FUNCTION_BLOCK TcaCarrier EXTENDS TcoCore.TcoComponent IMPLEMENTS ITcaCarrier
VAR CONSTANT
	MAX_WORKPIECEPLACES : INT := 127;
END_VAR

VAR PERSISTENT
	_carrierID : INT;	
	_data : TcaCarrierData;
	_config : TcaCarrierConfig;
	_arrayOfWorkpiecePlaces : ARRAY[0..MAX_WORKPIECEPLACES] OF TcaWorkpiecePlace(THIS^);
END_VAR

VAR
	_ModifyTask : TcaCarrierModifyTask(THIS^);	
	_modifyId : INT := 0;
	_i : INT;
		
	_WorkpieceStatusCount : ARRAY[0..eTcaWorkpiecePlaceStatus.MAXSIZE] OF INT;
	_PrimaryStatus : eTcaWorkpiecePlaceStatus;
	_SecondaryStatus : eTcaWorkpiecePlaceStatus;
	_PrimaryStatusCount : INT;
	_SecondaryStatusCount : INT;
	
	_ConfigError	: BOOL;
	
END_VAR

THIS^._ModifyTask(inoArrayOfWorkpiecePlaces := _arrayOfWorkpiecePlaces);

FOR _i:= 0 TO MAX_WORKPIECEPLACES DO
	_arrayOfWorkpiecePlaces[_i]();
END_FOR

METHOD ApplyConfig : REFERENCE TO TcaCarrier
VAR
	tmpData				: TcaCarrierConfig;
	
	tmpOffset 			: REAL;
	tmpOddRow			: INT;
	tmpEvenRow			: INT;
	tmpWorkpieceCount	: INT;
	
	tmpPos		 		: INT;
	tmpLoc		 		: INT;		
	tmpRow 				: INT;
	//tmpLvl				: INT;
	
	nRowNumber			: INT;
	nLocationNumber		: INT; 
	
	ni					: INT;
	
	tmpCoordinate 		: ST_Coordinate;		
END_VAR
tmpData := _config;

CASE tmpData.Layout OF
	eTcaCarrierLayout.Layout1 : 
		tmpOffset := 0;
		tmpOddRow := tmpData.PositionsInRow;
        tmpEvenRow := tmpData.PositionsInRow;
        tmpWorkpieceCount := tmpData.PositionsInRow*tmpData.PositionsInColumn;
		
    eTcaCarrierLayout.Layout2 :
		tmpOffset := 0.5;
		tmpOddRow := tmpData.PositionsInRow;
		tmpEvenRow := tmpData.PositionsInRow;
        tmpWorkpieceCount := tmpData.PositionsInRow*tmpData.PositionsInColumn;
		 
    eTcaCarrierLayout.Layout3 :
		 tmpOffset := -0.5;
		 tmpOddRow := tmpData.PositionsInRow;
         tmpEvenRow := tmpData.PositionsInRow;
         tmpWorkpieceCount := tmpData.PositionsInRow*tmpData.PositionsInColumn;	
		 
	eTcaCarrierLayout.Layout4 :
		 tmpOffset := -0.5;
		 tmpOddRow := tmpData.PositionsInRow;
         tmpEvenRow := tmpData.PositionsInRow + 1;
         tmpWorkpieceCount := tmpData.PositionsInRow*tmpData.PositionsInColumn + tmpData.PositionsInColumn/2;
		
	eTcaCarrierLayout.Layout5 :
		 tmpOffset := 0.5;
		 tmpOddRow := tmpData.PositionsInRow;
         tmpEvenRow := tmpData.PositionsInRow - 1;
         tmpWorkpieceCount := tmpData.PositionsInRow*tmpData.PositionsInColumn - tmpData.PositionsInColumn/2;
		 
END_CASE


MEMSET(ADR(_data.WorkpiecesCoordinate),0,SIZEOF(_data.WorkpiecesCoordinate));
MEMSET(ADR(_data.WorkpiecesEnabled),0,SIZEOF(_data.WorkpiecesEnabled));


FOR ni:= 0 TO tmpWorkpieceCount-1 DO
	
	// Bestimmen des Reihen und Spaltenndex und der x und y-Koordinate
	tmpPos := ni MOD tmpWorkpieceCount;
	tmpRow := tmpPos/(tmpOddRow + tmpEvenRow);	
	tmpLoc := tmpPos MOD (tmpOddRow + tmpEvenRow);
	
	IF tmpLoc >= tmpOddRow THEN
	    // gerade Reihe
	    nRowNumber := tmpRow*2 + 1;
	    nLocationNumber := tmpLoc - tmpOddRow;
	    tmpCoordinate.fX := tmpData.ColumnDistance*(nLocationNumber + tmpOffset)+tmpData.CoordinateFirstWorkpiece.fX;
	    tmpCoordinate.fY := tmpData.RowDistance*nRowNumber+tmpData.CoordinateFirstWorkpiece.fY;
	ELSE
	    // ungerade Reihe
	    nRowNumber := tmpRow*2;
	    nLocationNumber := tmpLoc;
	    tmpCoordinate.fX := tmpData.ColumnDistance*nLocationNumber+tmpData.CoordinateFirstWorkpiece.fX;
	    tmpCoordinate.fY := tmpData.RowDistance*nRowNumber+tmpData.CoordinateFirstWorkpiece.fY;
	END_IF
	
	tmpCoordinate.nOriginId := 0;
		
	_data.WorkpiecesCoordinate[ni] := tmpCoordinate;
	_data.WorkpiecesEnabled[ni] := TRUE;

END_FOR
END_METHOD

METHOD ChangeData : ITcoTaskStatus 
VAR_INPUT
	inData : TcaCarrierData;
END_VAR
ChangeData := _ModifyTask.InvokeCarrierData(inData);
END_METHOD

METHOD ColumnDistance : REFERENCE TO TcaCarrier
VAR_INPUT
	inDistance : LREAL;
END_VAR
THIS^._config.ColumnDistance:= inDistance;
ColumnDistance REF= THIS^;
END_METHOD

METHOD CoordinateFirstWorkpiece : REFERENCE TO TcaCarrier
VAR_INPUT
	inCoordinate : ST_Coordinate;
END_VAR
THIS^._config.CoordinateFirstWorkpiece:= inCoordinate;
CoordinateFirstWorkpiece REF= THIS^;
END_METHOD

METHOD CoordinatesOf : ST_Coordinate
VAR_INPUT
	WorkpiecePlace		: INT;
END_VAR

VAR
	tmpData				: TcaCarrierConfig;
	
	tmpOffset 			: REAL;
	tmpOddRow			: INT;
	tmpEvenRow			: INT;
	tmpWorkpieceCount	: INT;
	
	tmpPos		 		: INT;
	tmpLoc		 		: INT;		
	tmpRow 				: INT;
	//tmpLvl				: INT;
	
	nRowNumber			: INT;
	nLocationNumber		: INT; 
	
	tmpCoordinate 		: ST_Coordinate;		
	
END_VAR
IF WorkpiecePlace = 0 THEN
	RETURN;
END_IF

tmpData := _config;

CASE tmpData.Layout OF
	eTcaCarrierLayout.Layout1 : 
		tmpOffset := 0;
		tmpOddRow := tmpData.PositionsInRow;
        tmpEvenRow := tmpData.PositionsInRow;
        tmpWorkpieceCount := tmpData.PositionsInRow*tmpData.PositionsInColumn;
		
    eTcaCarrierLayout.Layout2 :
		tmpOffset := 0.5;
		tmpOddRow := tmpData.PositionsInRow;
		tmpEvenRow := tmpData.PositionsInRow;
        tmpWorkpieceCount := tmpData.PositionsInRow*tmpData.PositionsInColumn;
		 
    eTcaCarrierLayout.Layout3 :
		 tmpOffset := -0.5;
		 tmpOddRow := tmpData.PositionsInRow;
         tmpEvenRow := tmpData.PositionsInRow;
         tmpWorkpieceCount := tmpData.PositionsInRow*tmpData.PositionsInColumn;	
		 
	eTcaCarrierLayout.Layout4 :
		 tmpOffset := -0.5;
		 tmpOddRow := tmpData.PositionsInRow;
         tmpEvenRow := tmpData.PositionsInRow + 1;
         tmpWorkpieceCount := tmpData.PositionsInRow*tmpData.PositionsInColumn + tmpData.PositionsInColumn/2;
		
	eTcaCarrierLayout.Layout5 :
		 tmpOffset := 0.5;
		 tmpOddRow := tmpData.PositionsInRow;
         tmpEvenRow := tmpData.PositionsInRow - 1;
         tmpWorkpieceCount := tmpData.PositionsInRow*tmpData.PositionsInColumn - tmpData.PositionsInColumn/2;
		 
END_CASE

// Bestimmen des Reihen und Spaltenndex und der x und y-Koordinate
tmpPos := (WorkpiecePlace - 1) MOD tmpWorkpieceCount;
tmpRow := tmpPos/(tmpOddRow + tmpEvenRow);	
tmpLoc := tmpPos MOD (tmpOddRow + tmpEvenRow);
//tmpLvl := (Position - 1)/tmpWorkpieceCount;


IF tmpLoc >= tmpOddRow THEN
    // gerade Reihe
    nRowNumber := tmpRow*2 + 1;
    nLocationNumber := tmpLoc - tmpOddRow;
    tmpCoordinate.fX := tmpData.ColumnDistance*(nLocationNumber + tmpOffset);
    tmpCoordinate.fY := tmpData.RowDistance*nRowNumber;
ELSE
    // ungerade Reihe
    nRowNumber := tmpRow*2;
    nLocationNumber := tmpLoc;
    tmpCoordinate.fX := tmpData.ColumnDistance*nLocationNumber;
    tmpCoordinate.fY := tmpData.RowDistance*nRowNumber;
END_IF
		

//tmpCoordinate.fZ := tmpLvl*fLevelDistance;

// Koordinaten zurückgeben
tmpCoordinate.nOriginId := 0;
CoordinatesOf := tmpCoordinate;
END_METHOD

METHOD CountEmptyPlaces : INT

VAR
	tmp				: INT;
	ni				: INT;
END_VAR
CountEmptyPlaces := 0;

FOR ni := 0 TO MAX_WORKPIECEPLACES DO
	
	IF NOT _arrayOfWorkpiecePlaces[ni].Enabled THEN
		CONTINUE;
	END_IF
	
	IF _arrayOfWorkpiecePlaces[ni].Error THEN
		CONTINUE;
	END_IF

	IF NOT _arrayOfWorkpiecePlaces[ni].WorkpiecePresent THEN
		tmp := tmp + 1;	
	END_IF

END_FOR

CountEmptyPlaces := tmp;
END_METHOD

METHOD CountPlacesByStatus : INT
VAR_INPUT
	nStatus			: INT;
END_VAR

VAR
	tmp				: INT;
	ni				: INT;
END_VAR
CountPlacesByStatus := 0;

FOR ni := 0 TO MAX_WORKPIECEPLACES DO

	IF NOT _data.WorkpiecesData[ni].Enabled THEN
		CONTINUE;
	END_IF	
	
	IF _data.WorkpiecesData[ni].Error THEN
		CONTINUE;
	END_IF

	IF _data.WorkpiecesData[ni].CurrentStatus = nStatus THEN
			tmp := tmp + 1;
	END_IF
	
END_FOR

CountPlacesByStatus := tmp;
END_METHOD

PROPERTY Data : REFERENCE TO TcaCarrierData
GET
Data REF= _data;
END_GET
END_PROPERTY

//FB_Init ist immer implizit verfügbar und wird primär für die Initialisierung verwendet.
//Der Rückgabewert wird nicht ausgewertet. Für gezielte Einflussnahme können Sie
//die Methoden explizit deklarieren und darin mit dem Standard-Initialisierungscode 
//zusätzlichen Code bereitstellen. Sie können den Rückgabewert auswerten.
METHOD FB_Init: BOOL
VAR_INPUT    
bInitRetains: BOOL; // TRUE: Die Retain-Variablen werden initialisiert (Reset warm / Reset kalt)    
bInCopyCode: BOOL;  // TRUE: Die Instanz wird danach in den Kopiercode kopiert (Online-Change)
ParentObject : ITcoObject;
END_VAR
VAR
	_i : INT;
END_VAR
FOR _i:= 0 TO MAX_WORKPIECEPLACES DO
	_arrayOfWorkpiecePlaces[_i].Id := _i+1;
END_FOR

RETURN;
END_METHOD

METHOD FillWithWorkpieces_CustomStatus : ITcoTaskStatus
VAR_INPUT
	Status		: eTcaWorkpiecePlaceStatus;
END_VAR
FillWithWorkpieces_CustomStatus := _ModifyTask.InvokeWorkpieceCommand(eTcaCarrierCmd.fillPlaces, Status);
END_METHOD

METHOD FillWithWorkpieces_InitialStatus : ITcoTaskStatus
VAR_INPUT
END_VAR
IF _data.RequestStatus = eTcaWorkpiecePlaceStatus.undefined THEN
	RETURN;
END_IF

FillWithWorkpieces_InitialStatus := _ModifyTask.InvokeWorkpieceCommand(eTcaCarrierCmd.fillPlaces, _data.InitialStatus);
END_METHOD

{attribute 'TcRpcEnable'}
METHOD FillWithWorkpieces_RequestStatus : ITcoTaskStatus
VAR_INPUT
END_VAR
IF Data.RequestStatus = eTcaWorkpiecePlaceStatus.undefined THEN
	RETURN;
END_IF

FillWithWorkpieces_RequestStatus := _ModifyTask.InvokeWorkpieceCommand(eTcaCarrierCmd.fillPlaces, Data.RequestStatus);
END_METHOD

METHOD FindPlace : REFERENCE TO TcaWorkpiecePlace //-1..no Position found

VAR_INPUT
	Status		: eTcaWorkpiecePlaceStatus;
END_VAR

VAR
	ni				: INT;
END_VAR
FindPlace REF= 0;
FOR ni := 0 TO MAX_WORKPIECEPLACES DO
	
	IF NOT _data.WorkpiecesData[ni].Enabled THEN
		CONTINUE;
	END_IF	
	
	IF _data.WorkpiecesData[ni].Error THEN
		CONTINUE;
	END_IF	

	IF _data.WorkpiecesData[ni].CurrentStatus = Status OR Status < eTcaWorkpiecePlaceStatus.undefined THEN
	   
		FindPlace REF= _arrayOfWorkpiecePlaces[ni];
		EXIT;
		
	END_IF	
END_FOR
END_METHOD

METHOD GetPlaceReference : REFERENCE TO TcaWorkpiecePlace
VAR_INPUT
	nIndexNr		: INT;
END_VAR
IF nIndexNr < 0 OR nIndexNr > MAX_WORKPIECEPLACES THEN
	RETURN;
END_IF

GetPlaceReference REF= _arrayOfWorkpiecePlaces[nIndexNr];
END_METHOD

PROPERTY InitialStatus : eTcaWorkpiecePlaceStatus
GET
InitialStatus := _data.InitialStatus;
END_GET
SET
_data.InitialStatus := InitialStatus;
END_SET
END_PROPERTY

METHOD Layout : REFERENCE TO TcaCarrier
VAR_INPUT
	inLayout : eTcaCarrierLayout;
END_VAR
THIS^._config.Layout:= inLayout;
Layout REF= THIS^;
END_METHOD

PROPERTY ModifyTask : TcoCore.ITcoTaskStatus
GET
ModifyTask := _ModifyTask;
END_GET
END_PROPERTY

METHOD PositionsInColumn : REFERENCE TO TcaCarrier
VAR_INPUT
	inPositionsInColumn : INT;
END_VAR
THIS^._config.PositionsInColumn:= inPositionsInColumn;
PositionsInColumn REF= THIS^;
END_METHOD

METHOD PositionsInRow : REFERENCE TO TcaCarrier
VAR_INPUT
	inPositionsInRow : INT;
END_VAR
THIS^._config.PositionsInRow:= inPositionsInRow;
PositionsInRow REF= THIS^;
END_METHOD

METHOD RefreshStatus : BOOL
VAR
	ni			: INT;
END_VAR
MEMSET(ADR(_WorkpieceStatusCount), 0, SIZEOF(_WorkpieceStatusCount));
_data.InitialStatus := eTcaWorkpiecePlaceStatus.undefined;
_data.RequestStatus := eTcaWorkpiecePlaceStatus.undefined;

FOR ni := 0 TO MAX_WORKPIECEPLACES DO
	
	IF NOT _arrayOfWorkpiecePlaces[ni].Enabled THEN
		CONTINUE;
	END_IF

		
	IF _data.WorkpiecesData[ni].CurrentStatus = eTcaWorkpiecePlaceStatus.undefined THEN
		CONTINUE;
	END_IF

	_WorkpieceStatusCount[_data.WorkpiecesData[ni].CurrentStatus] := _WorkpieceStatusCount[_data.WorkpiecesData[ni].CurrentStatus] + 1;
	
	IF _WorkpieceStatusCount[_data.WorkpiecesData[ni].CurrentStatus] >= _WorkpieceStatusCount[_PrimaryStatus] THEN
		_SecondaryStatus := _PrimaryStatus;
		_PrimaryStatus := _data.WorkpiecesData[ni].CurrentStatus;
	END_IF

END_FOR


IF _PrimaryStatus = _SecondaryStatus THEN
	_SecondaryStatus := 0;
END_IF

_modifyId := _modifyId + 1;
END_METHOD

PROPERTY RequestStatus : eTcaWorkpiecePlaceStatus
GET
RequestStatus := _data.RequestStatus;
END_GET
SET
_data.RequestStatus := RequestStatus;
END_SET
END_PROPERTY

(*~
	<docu>
		<summary>
			Restores this instance to the Ready state. Can be called explicitly or from within one of the restore mechanisms.	
		</summary>			
	</docu>	
~*)
METHOD Restore : TcoCore.ITcoRestorable

VAR
	_i : INT;
END_VAR
FOR _i:= 0 TO MAX_WORKPIECEPLACES DO
	_arrayOfWorkpiecePlaces[_i].Restore();
END_FOR

RefreshStatus();
END_METHOD

METHOD RowDistance : REFERENCE TO TcaCarrier
VAR_INPUT
	inDistance : LREAL;
END_VAR
THIS^._config.RowDistance:= inDistance;
RowDistance REF= THIS^;
END_METHOD

(*~
	<docu>
		<summary>
		    Custom service (manual, maintenance) logic.
			This method must be implemented in derived class.
		</summary>			
	</docu>	
~*)
METHOD PROTECTED ServiceMode
VAR
	_i : INT;
END_VAR
FOR _i:= 0 TO MAX_WORKPIECEPLACES DO
	_arrayOfWorkpiecePlaces[_i].Service();
END_FOR
END_METHOD

PROPERTY Task : TcoCore.ITcoTask
GET
Task := _ModifyTask;
END_GET
END_PROPERTY

PROPERTY WorkpiecePlaces : INT
GET
CASE _config.Layout OF	
	eTcaCarrierLayout.Layout1 : WorkpiecePlaces := _config.PositionsInRow*_config.PositionsInColumn;		
    eTcaCarrierLayout.Layout2 : WorkpiecePlaces := _config.PositionsInRow*_config.PositionsInColumn;		 
    eTcaCarrierLayout.Layout3 : WorkpiecePlaces := _config.PositionsInRow*_config.PositionsInColumn;		 
	eTcaCarrierLayout.Layout4 : WorkpiecePlaces := _config.PositionsInRow*_config.PositionsInColumn + _config.PositionsInColumn/2;		
	eTcaCarrierLayout.Layout5 : WorkpiecePlaces := _config.PositionsInRow*_config.PositionsInColumn - _config.PositionsInColumn/2;		
	ELSE
		 WorkpiecePlaces := 0;
END_CASE
END_GET
END_PROPERTY

END_FUNCTION_BLOCK

(* stored: Version 1.1.0.1
   POU TcaCarrier: Id {cb4cb05c-8cc6-4c4e-b4d4-2bd8871ee7cb}, SpecialFunc None
   Folder Config: Id {5b12d6a7-75e3-4cf0-aa63-45d3948de01c}
   Folder Functions: Id {e179f35a-15b1-4e1d-a2be-a3074b0e5c68}
   Folder Operations: Id {56bebb71-64cc-4645-900b-db953e179838}
   Method ApplyConfig: Id {ec2ab732-0b05-4cd8-9ee3-ccd0e42fc7dd}
   Method ChangeData: Id {37e814ce-5f8e-4579-82af-1e56bc0379a9}
   Method ColumnDistance: Id {061779de-a8a4-4f45-bbe5-36d216596b95}
   Method CoordinateFirstWorkpiece: Id {b9aec3d5-66bd-4a01-a556-8878c2af4d3e}
   Method CoordinatesOf: Id {fb9ca07f-d465-4155-b936-ffa9ed3dcdea}
   Method CountEmptyPlaces: Id {180bc4e3-ba20-47fb-92c1-8b8a99e6818d}
   Method CountPlacesByStatus: Id {d8fa782e-a592-4393-b541-142317da77e8}
   Property Data: Id {14535b80-8544-4b5c-b46c-52fec6e6c4f6}
   Get Get: Id {8f511891-98a7-4369-8bb4-605ff91c3d4e}
   Method FB_Init: Id {a39378d3-a146-42e4-81d7-513f20fa6674}
   Method FillWithWorkpieces_CustomStatus: Id {3b0c22c0-d494-4035-843c-f65b12875767}
   Method FillWithWorkpieces_InitialStatus: Id {8f51a660-10db-4072-8773-021604a9acb8}
   Method FillWithWorkpieces_RequestStatus: Id {41c8d7c9-26de-4ec8-80c0-2da1719e22de}
   Method FindPlace: Id {6021ca1e-a1ef-4ea5-9e46-c898a3806339}
   Method GetPlaceReference: Id {c781c58b-59de-49f8-ac75-8ffb97aab0ac}
   Property InitialStatus: Id {bf6848df-442f-4b63-9f1d-fe6a13da345e}
   Get Get: Id {9da4bb88-8967-4f68-a769-9abfaf59e8ef}
   Set Set: Id {013a6002-b5d6-4353-8b59-74a706e2aed7}
   Method Layout: Id {3b05a680-4427-40f2-baf3-c7000d9bb89c}
   Property ModifyTask: Id {b22af8ee-20cc-436b-969e-549731099c33}
   Get Get: Id {bf44bf0d-eaa6-4038-a146-905b63014044}
   Method PositionsInColumn: Id {7377dbc3-f6fd-42e2-8707-de70abea79c5}
   Method PositionsInRow: Id {1465c2a1-a580-4c76-a912-36bd2f7017f1}
   Method RefreshStatus: Id {45b28ecb-4270-41ad-aa1b-7502953923ca}
   Property RequestStatus: Id {a9d116ea-9b1e-4fa9-9bc2-641207b5540c}
   Get Get: Id {13d13370-6282-4360-bfec-38b264fb8263}
   Set Set: Id {ecc5f7c6-ef16-4cc4-bfe9-d4529123d750}
   Method Restore: Id {3b14de8e-b3fb-407e-8523-ab59c2b6b5a1}
   Method RowDistance: Id {d7fbb5a1-34c6-43ca-ad90-adfacf90b230}
   Method ServiceMode: Id {210a8b18-6f62-4d7f-977f-4f3cf935d237}
   Property Task: Id {37cb437b-8616-4f31-b387-1db1769d082a}
   Get Get: Id {15638a30-b372-459a-96e3-0012ed9625d7}
   Property WorkpiecePlaces: Id {4743c045-c7f1-4ea2-877a-78415e57eca8}
   Get Get: Id {1b62398e-be48-4c80-8efa-d02ec467eb4d} *)
